FUNCTION_BLOCK FB_ROS2Skill EXTENDS FB_Skill
VAR_INPUT
	{attribute 'OPC.UA.DA.StructuredType':=1}
	{attribute 'OPC.UA.DA' := '1'}
	Control     : ST_SkillControl;
	{attribute 'OPC.UA.DA.StructuredType':=1}
	{attribute 'OPC.UA.DA' := '1'}
    Status      : ST_SkillStatus;

//     Specific    : ST_RobotMoveSpecific;
	
END_VAR
VAR_OUTPUT
END_VAR
VAR
END_VAR

{warning 'Add property implementation'}
PROPERTY Busy : BOOL
GET
IF _state=eState.Active THEN
	Busy:=TRUE;
ELSE
	Busy:=FALSE;
END_IF
END_GET
END_PROPERTY

// {error 'Add property implementation or delete property to use base implementation'}
PROPERTY Done : BOOL
GET
END_GET
END_PROPERTY

METHOD onActivate : BOOL
// ---- Init ----
transitionresult:=eResult.None;



// ---- Change ----




// ---- Check ----
transitionresult := eResult.SUCCESS;


// ---- Change State ----
IF transitionresult= eResult.SUCCESS THEN
	State:=eState.Active;
ELSIF transitionresult= eResult.FAILURE THEN
	State:=eState.Inactive;
ELSIF transitionresult= eResult.ERROR THEN
	State:=eState.ErrorProcessing;
ELSE
	ADSLOGSTR(ADSLOG_MSGTYPE_WARN,'Transitionresult from onActivate is None','');
END_IF
END_METHOD

METHOD onCleanup : BOOL
// ---- Init ----
transitionresult:=eResult.None;



// ---- Change ----



// ---- Check ----
transitionresult := eResult.SUCCESS;


// ---- Change State ----
IF transitionresult= eResult.SUCCESS THEN
	State:=eState.Unconfigured;
ELSIF transitionresult= eResult.FAILURE THEN
	ADSLOGSTR(ADSLOG_MSGTYPE_WARN,'Transitionresult from onCleanup is FAILURE ','');
ELSIF transitionresult= eResult.ERROR THEN
	State:=eState.ErrorProcessing;
ELSE
	ADSLOGSTR(ADSLOG_MSGTYPE_WARN,'Transitionresult from onCleanup is NONE','');
END_IF
END_METHOD

METHOD onConfigure : BOOL
// ---- Init ----
transitionresult:=eResult.None;



// ---- Change ----


// ---- Check ----
transitionresult := eResult.SUCCESS;


// ---- Change State ----
IF transitionresult= eResult.SUCCESS THEN
	State:=eState.Inactive;
ELSIF transitionresult= eResult.FAILURE THEN
	State:=eState.Unconfigured;
ELSIF transitionresult= eResult.ERROR THEN
	State:=eState.ErrorProcessing;
ELSE
	ADSLOGSTR(ADSLOG_MSGTYPE_WARN,'Transitionresult from onConfigure is None','');
END_IF
END_METHOD

METHOD onDeactivate : BOOL
// ---- Init ----
transitionresult:=eResult.None;



// ---- Change ----
 //Stopping SFC



// ---- Check ----
transitionresult := eResult.SUCCESS;


// ---- Change State ----
IF transitionresult= eResult.SUCCESS THEN
	State:=eState.Inactive;
ELSIF transitionresult= eResult.FAILURE THEN
	ADSLOGSTR(ADSLOG_MSGTYPE_WARN,'Transitionresult from onDeactivate is FAILURE','');
ELSIF transitionresult= eResult.ERROR THEN
	State:=eState.ErrorProcessing;
ELSE
	ADSLOGSTR(ADSLOG_MSGTYPE_WARN,'Transitionresult from onDeactivate is None','');
END_IF
END_METHOD

METHOD onError : BOOL
// ---- Init ----
transitionresult:=eResult.None;



// ---- Change ----





// ---- Check ----
transitionresult := eResult.SUCCESS;


// ---- Change State ----
IF transitionresult= eResult.SUCCESS THEN
	State:=eState.Unconfigured;
ELSIF transitionresult= eResult.FAILURE THEN
	State:=eState.Finalized;
ELSIF transitionresult= eResult.ERROR THEN
	ADSLOGSTR(ADSLOG_MSGTYPE_WARN,'Transitionresult from onError is Error','');
ELSE
	ADSLOGSTR(ADSLOG_MSGTYPE_WARN,'Transitionresult from onError is None','');
END_IF
END_METHOD

METHOD onShutdown : BOOL
// ---- Init ----
transitionresult:=eResult.None;



// ---- Change ----



// ---- Check ----
transitionresult := eResult.SUCCESS;


// ---- Change State ----
IF transitionresult= eResult.SUCCESS THEN
	State:=eState.Finalized;
ELSIF transitionresult= eResult.FAILURE THEN
	ADSLOGSTR(ADSLOG_MSGTYPE_WARN,'Transitionresult from onShutdown is FAILURE','');
ELSIF transitionresult= eResult.ERROR THEN
	State:=eState.ErrorProcessing;
ELSE
	ADSLOGSTR(ADSLOG_MSGTYPE_WARN,'Transitionresult from onShutdown is None','');
END_IF
END_METHOD

METHOD Pause : BOOL
Control.Pause:=True;
END_METHOD

METHOD Restart : BOOL
Stop();
Start();
END_METHOD

METHOD Resume : BOOL
END_METHOD

METHOD Start : BOOL
Control.Start:=True;
END_METHOD

METHOD Stop : BOOL
Control.Cancel:=True;
END_METHOD

END_FUNCTION_BLOCK

(* stored: Version 1.1.0.1, ProductVersion 3.1.4026.18
   POU FB_ROS2Skill: Id {2e00d6a1-8d22-4bf8-a533-217a1a8bd953}, SpecialFunc None
   Folder StateControl: Id {a0d7267b-99f4-41f2-8af1-fa0fbdfbdb62}
   Property Busy: Id {09e5b3c9-ee64-44a2-abd8-5d4d03bc4b38}
   Get Get: Id {b2f257ba-29de-49be-8325-f1b3106f7d1e}
   Property Done: Id {050d33ac-91a8-488e-bf4c-71a63756542c}
   Get Get: Id {b8d8e9c2-e134-4622-b2f9-fa8db2321a8a}
   Method onActivate: Id {bc2d83b7-2512-4688-a8e1-54e2299564c4}
   Method onCleanup: Id {6fd91c29-8e32-488f-9ae6-151d92027456}
   Method onConfigure: Id {d115cc8e-7f1a-49b5-899a-a8343b56dd26}
   Method onDeactivate: Id {88519088-d0f4-44de-be30-f5617d391955}
   Method onError: Id {6f028444-e95e-464c-8fca-f4509fc4038a}
   Method onShutdown: Id {46466cbc-d126-42d4-a4a0-92feae79e9e1}
   Method Pause: Id {1e98ec14-2d0f-46f1-beaa-7c0329f01f5f}
   Method Restart: Id {e4adb370-5ab1-4ddd-867f-399f400037c2}
   Method Resume: Id {5817404e-7120-47d3-bfe5-80fb599fffeb}
   Method Start: Id {2cb6dfed-a48a-423f-8932-7f6194b92564}
   Method Stop: Id {23b5ab90-30ca-487b-9c78-f9423fb9e265} *)
